// TIA Portal V16 export
// export: Created 2021-09-02T13:55:53.4783388Z, ExportSetting WithDefaults, DisplayName Totally Integrated Automation Portal, DisplayVersion V16 Update 3, DisplayName TIA Portal Version Control Interface, DisplayVersion V16 Update 2, DisplayName TIA Portal Openness, DisplayVersion V16 Update 3, DisplayName TIA Portal Teamcenter Gateway, DisplayVersion V16, DisplayName STEP 7 Professional, DisplayVersion V16 Update 3, DisplayName STEP 7 Safety, DisplayVersion V16, DisplayName WinCC Advanced, DisplayVersion V16 Update 3
TYPE "Sequence"
// stored: IsFailsafeCompliant false
   STRUCT
      devOn : Array["MIN_STEP_NUMB".."MAX_STEP_NUMB", "MIN_DEV_NUMB".."MAX_DEV_NUMB"] of Bool;
      delay : Array["MIN_STEP_NUMB".."MAX_STEP_NUMB"] of Int;
   END_STRUCT;
   // devOn[1,1] := TRUE;
   // delay[1..3] := 1;
END_TYPE
